TEXTLIST TextList_SubTankerroid
  0 = 'no_error'
  1 = 'pump_timeout'
  2 = 'back_to_air_tank'
  666 = 'emergency_error'
   = ''
END_TEXTLIST

(* stored: Version 1.1.0.1, ProductVersion 3.1.4024.11
   TextList TextList_SubTankerroid: Id {67168a1e-ee7f-436c-9ce3-6b76a723958b} *)
